{attribute 'GeneratedUsingTerminal: EL6201-0000-0017'}
{attribute addProperty BoxType "EL6201-0000-0017"}
{attribute addProperty Id "Slave_14A_DO0BOOL1Slave_14A_DO1BOOL1Slave_14A_DO2BOOL1Slave_14A_DO3BOOL1Slave_14B_DO0BOOL1Slave_14B_DO1BOOL1Slave_14B_DO2BOOL1Slave_14B_DO3BOOL1"}
{attribute addProperty CRC "1290242747"}
{attribute addProperty Size "8"}
TYPE Slave_14_Outputs_4CE78ABB :
STRUCT
	{attribute addProperty Name "Slave_14A_DO0"}
	Slave_14A_DO0 : BOOL;
	{attribute addProperty Name "Slave_14A_DO1"}
	Slave_14A_DO1 : BOOL;
	{attribute addProperty Name "Slave_14A_DO2"}
	Slave_14A_DO2 : BOOL;
	{attribute addProperty Name "Slave_14A_DO3"}
	Slave_14A_DO3 : BOOL;
	{attribute addProperty Name "Slave_14B_DO0"}
	Slave_14B_DO0 : BOOL;
	{attribute addProperty Name "Slave_14B_DO1"}
	Slave_14B_DO1 : BOOL;
	{attribute addProperty Name "Slave_14B_DO2"}
	Slave_14B_DO2 : BOOL;
	{attribute addProperty Name "Slave_14B_DO3"}
	Slave_14B_DO3 : BOOL;
END_STRUCT
END_TYPE

(* stored: Version 1.2.0.0, ProductVersion 3.1.4024.9
   DUT Slave_14_Outputs_4CE78ABB: Id {0ab1b433-1234-4207-9a2d-001e8be68e15} *)
